(* PLC project Tc2_Standard.CTUD Demo, tc3-libraries-kb TwinCAT 3.1 *)
(* stored: creationDateTime 2026-05-10T08:00:00, modificationDateTime 2026-05-10T08:00:00 *)

PROGRAM P_Demo_CTUD
  VAR
    fbCTUD : CTUD;  (* Counter 实例 *)
    bIn : BOOL;  (* 进料：CV+1 *)
    bOut : BOOL;  (* 出料：CV-1 *)
    bReset : BOOL;  (* 清零 *)
    bLoad : BOOL;  (* 装入满库 8 件 *)
    bFull : BOOL;  (* 已满 (CV >= 8) *)
    bEmpty : BOOL;  (* 已空 (CV = 0) *)
    nCV : WORD;  (* 当前库存 *)
  END_VAR

            // ============================================================
// Tc2_Standard.CTUD 演示程序
// ============================================================
// 场景：进料增计数、出料减计数，限位 8 件库存
// 验证步骤：
//   1. 把本 PROGRAM 加到 PlcTask 调用列表
//   2. 编译并登录目标
//   1. bReset 一次 → nCV = 0、bEmpty = TRUE
//   2. bIn 上升沿 8 次 → nCV = 8、bFull = TRUE
//   3. bOut 上升沿 8 次 → nCV = 0、bEmpty = TRUE
//   4. bLoad 一次 → nCV = 8、bFull = TRUE（一键装满）
// ============================================================

fbCTUD(
    CU    := bIn,
    CD    := bOut,
    RESET := bReset,
    LOAD  := bLoad,
    PV    := WORD#8,
    QU    => bFull,
    QD    => bEmpty,
    CV    => nCV
);

          
END_PROGRAM
